REGION Network 18: Special characters — Common character widths and additional whitespace characters
   // ▀▀▀▀▀▀▀▀▀▀▀▀▀▀▀▀▀▀▀▀▀▀▀▀▀▀▀▀▀▀▀▀▀▀▀▀▀▀▀▀▀▀▀▀
   // 
   // TITLE:    COMMON CHARACTER WIDTHS AND ADDITIONAL WHITESPACE CHARACTERS
   // 
   // ▄▄▄▄▄▄▄▄▄▄▄▄▄▄▄▄▄▄▄▄▄▄▄▄▄▄▄▄▄▄▄▄▄▄▄▄▄▄▄▄▄▄▄▄
   // 
   // 
   // This section contains a list of the alphanumeric characters and common punctuation in terms of
   // character width (thinnest first).
   // 
   // The average character widths for each group are based on the frequency of letter usage in 
   // standard (British) English.
   // 
   // The additional whitespace characters complete the set of TIA Portal whitespace characters, these
   // are included for completeness, but duplicate the widths of the standard whitespace characters 
   // listed in previous sections.
   // 
   // 
   // 
   // ▄▄▄▄▄▄▄▄▄▄▄▄▄▄▄▄▄▄▄▄▄▄▄▄▄▄▄▄▄▄▄▄▄▄▄▄▄▄▄▄▄▄▄▄
   // NORMAL CHARACTERS BY WIDTH
   // 
   // 
   // ▐I▌1sp
   // ▐J▌1⅓ sp
   // ▐T▌1⅔ SP
   // ▐F▌2 sp
   // ▐L▌2 sp
   // ▐P▌2 sp
   // ▐R▌2 sp
   // ▐A▌2⅓ SP
   // ▐B▌2⅓ SP
   // ▐C▌2⅓ SP
   // ▐E▌2⅓3 SP
   // ▐K▌2⅓ SP
   // ▐S▌2⅓ SP
   // ▐V▌2⅓ SP
   // ▐X▌2⅓ SP
   // ▐Y▌2⅓ SP
   // ▐Z▌2⅓ SP
   // ▐D▌2⅔ sp
   // ▐G▌2⅔ sp
   // ▐H▌2⅔ sp
   // ▐N▌2⅔ sp
   // ▐U▌2⅔ sp
   // ▐M▌3 sp
   // ▐O▌3 sp
   // ▐Q▌3 sp
   // ▐W▌3 sp
   // Upper avg. (based on frequency and width) = 2.25 normal spaces
   // 
   // ▐f▌1 sp
   // ▐i▌1 sp
   // ▐j▌1 sp
   // ▐l▌1 sp
   // ▐r▌1⅓ sp
   // ▐t▌1⅓ sp
   // ▐x▌1⅔ sp
   // ▐y▌1⅔ sp
   // ▐z▌1⅔ sp
   // ▐c▌2 sp
   // ▐k▌2 sp
   // ▐s▌2 sp
   // ▐v▌2 sp
   // ▐a▌2⅓ sp
   // ▐b▌2⅓ sp
   // ▐d▌2⅓ sp
   // ▐e▌2⅓ sp
   // ▐g▌2⅓ sp
   // ▐h▌2⅓ sp
   // ▐n▌2⅓ sp
   // ▐o▌2⅓ sp
   // ▐p▌2⅓ sp
   // ▐q▌2⅓ sp
   // ▐u▌2⅓ sp
   // ▐w▌3 sp
   // ▐m▌3⅔ sp
   // Lower avg. (based on frequency and width) = 2.00 normal spaces
   // 
   // ▐0▌2⅓ sp
   // ▐1▌2⅓ sp
   // ▐2▌2⅓ sp
   // ▐3▌2⅓ sp
   // ▐4▌2⅓ sp
   // ▐5▌2⅓ sp
   // ▐6▌2⅓ sp
   // ▐7▌2⅓ sp
   // ▐8▌2⅓ sp
   // ▐9▌2⅓ sp
   // Numbers = 2.33 sp
   // 
   // ▐!▌1 sp
   // ▐'▌1 sp
   // ▐,▌1 sp
   // ▐-▌1 sp
   // ▐.▌1 sp
   // ▐/▌1 sp
   // ▐\▌1 sp
   // ▐|▌1 sp
   // ▐[▌1⅓ sp
   // ▐]▌1⅓ sp
   // ▐:▌1⅓ sp
   // ▐:▌1⅓ sp
   // ▐(▌1⅓ sp
   // ▐)▌1⅓ sp
   // ▐{▌1⅔ sp
   // ▐}▌1⅔ sp
   // ▐"▌1⅔ sp
   // ▐?▌1⅔ sp
   // ▐<▌2 sp
   // ▐>▌2 sp
   // ▐^▌2 sp
   // ▐_▌2 sp
   // ▐~▌2 sp
   // ▐=▌2⅓ sp
   // ▐$▌2⅓ sp
   // ▐*▌2⅓ sp
   // ▐+▌2⅓ sp
   // ▐`▌2⅓ sp
   // ▐&▌2⅔ sp
   // ▐#▌2⅔ sp
   // ▐%▌3 sp
   // ▐@▌3⅓ sp
   // Punctuation avg. 1 sp (based on comma, full stop and dash being the most common)
   // 
   // 
   // 
   // ▄▄▄▄▄▄▄▄▄▄▄▄▄▄▄▄▄▄▄▄▄▄▄▄▄▄▄▄▄▄▄▄▄▄▄▄▄▄▄▄▄▄▄▄
   // ALL OTHER WHITESPACE CHARACTERS
   // 
   // The other whitespace characters (Hair space, figure space &c.) are supported by the Siemens
   // font, but have the identical widths to those listed above. The full list is shown below:
   // 
   // ▐  ▌2 Em spaces
   // ▐    ▌4 En space      (1/2 em)
   // ▐      ▌6 Three per em     (1/3 em)
   // ▐        ▌8 Punctuation space (1/4 em)
   // ▐        ▌8 Normal space      (1/4 em)
   // ▐        ▌8 Four per em      (1/4 em)
   // ▐        ▌8 Figure space     (1/4 em)
   // ▐            ▌12 Six per em    (1/6 em)
   // ▐            ▌12 Hair space       (1/6 em)
   // 
   //                 ━━━  ⬙⬙⬙⬙⬙⬙  ━━━
   // 
   // 
   // ██████████████ █ █ █ █  END   █ █ █ █ ██████████████
END_REGION

REGION Network 19: OB1 NETWORK 1 — Project description
   // ▀▀▀▀▀▀▀▀▀▀▀▀▀▀▀▀▀▀▀▀▀▀▀▀▀▀▀▀▀▀▀▀▀▀▀▀▀▀▀▀▀▀▀▀
   // 
   // TITLE:    PS2001 — PRACTICAL SERIES AUTOMATION LIBRARY
   // 
   // ▄▄▄▄▄▄▄▄▄▄▄▄▄▄▄▄▄▄▄▄▄▄▄▄▄▄▄▄▄▄▄▄▄▄▄▄▄▄▄▄▄▄▄▄
   // 
   // 
   // ――――――――――――――――――――――――――――――――――
   // COPYRIGHT:       © 2020 Michael Gledhill
   //           Part of the Practical Series of Publications
   //           Published in the United Kingdom
   //           mg@practicalseries.com
   //           https://practicalseries.com
   // ――――――――――――――――――――――――――――――――――
   // CUSTOMER:       Practical Series of Publications (PSP)
   // 
   // PROJECT:      Practical Series Automation Library (PAL)
   // 
   // PROJECT NO.:       PS2001
   // ――――――――――――――――――――――――――――――――――
   // CONTROLLER:       CPU 1515-2PN/DP
   // 
   // CONTROLLER NAME:    CON100
   // 
   // IP ADDRESS:      192.168.001.100
   // ――――――――――――――――――――――――――――――――――
   // TIA PROJECT NAME:    PS2001-PAL-D0000
   // 
   // STATUS:        DEVELOPMENT
   // ――――――――――――――――――――――――――――――――――
   // PROTECTION:     To minimise the risk of inadvertent modification to 
   //           tested modules, certain blocks will be released for 
   //           use with “protected access” (referred to a “write 
   //           protection” in Siemens terminology), this allows the 
   //           block to be used normally, but prevents the block 
   //           being accidentally modified. 
   // 
   //           This is in accordance with the risk assessment given 
   //           in the Validation Plant (VP), Appendix A [Ref. 002].
   // 
   //           ┌─────────────────────┐
   //           │ THE WRITE PROTECTION PASSWORD IS: PS2001 │
   //           └─────────────────────┘
   // 
   // 
   // ▄▄▄▄▄▄▄▄▄▄▄▄▄▄▄▄▄▄▄▄▄▄▄▄▄▄▄▄▄▄▄▄▄▄▄▄▄▄▄▄▄▄▄▄
   // PROJECT OVERVIEW
   // 
   // 
   // The PAL is a library of software modules and templates that have been developed for the 
   // Siemens Simatic S7-1500 range of controllers (and to a lesser extent the S7-1200 range).
   // 
   // The full library and all necessary documentation is available from the Practical Series website:
   // 
   //      https://practicalseries.com/2001-pal/index.html
   // 
   // 
   // The PAL is configured and deployed using the Siemens Simatic TIA Portal programming 
   // environment.
   // 
   // The PAL software structure is designed such that it is applicable to virtually all industrial 
   // applications that can generally controlled by a programmable logic controller.
   // 
   // The PAL software being developed as part of this Project, is considered to be suitable for use in 
   // the following types of industries (this is not an exhaustive list):
   // 
   //    •   Water and waste water treatment
   //    •   Pharmaceutical and batch production
   //    •   Brewing and fermentation
   //    •   Chemical manufacturing
   //    •   Oil and gas systems
   //    •   Food and beverage production
   // 
   // Such applications can generally be thought of as processes that operate with a response time
   // of more than 100 ms. I.e. the system would not be expected to respond to some stimuli faster
   // than 100 ms. In practice, a Controller may (and usually will) respond faster than this; however, 
   // a response time of 100 ms is considered to be an acceptable limit for PLC control.
   // 
   // At its most basic level, the PAL will be a library of software modules that control the fundamental 
   // aspects of an industrial plant; such modules would for example read the value of an instrument, 
   // operate a valve or drive, perform a calculation &c.
   // 
   // Such software modules are referred to as standard modules, these are fixed modules that 
   // perform a particular function and are identical across all software installations.
   // 
   // The PAL also contains application specific modules; these contain software that is applicable 
   // to the plant being controlled.
   // 
   // The Practical Series Automation Library is freely available under the MIT Open Source licence 
   // (see below). Those who find it useful may, if they wish, make a donation to support the library. 
   // 
   // Donations can be made here:
   // 
   //      https://practicalseries.com/2001-pal/11-web/81-00-pay.html
   // 
   // The PAL contains fully deployable software that has been developed by the author in his 
   // profession as a chartered electrical engineer. It is currently in use on various live plants 
   // throughout the UK and in some other parts of the world. 
   // 
   // This software is suitable for controlling and automating most industrial applications (typical 
   // process applications). It is easy to use and configure, but does have a degree of practical 
   // complexity appropriate for the environments within which it is employed. It is heavily 
   // configurable, has various operating modes and is suitable for a multitude of industrial 
   // applications.
   // 
   // IF YOU DON’T UNDERSTAND IT, DON’T USE IT. IF YOU DO USE IT, YOU DO SO AT YOUR OWN RISK.
   // 
   //                ━━━   ⬙⬙⬙⬙⬙⬙   ━━━
   // 
   // ▄▄▄▄▄▄▄▄▄▄▄▄▄▄▄▄▄▄▄▄▄▄▄▄▄▄▄▄▄▄▄▄▄▄▄▄▄▄▄▄▄▄▄▄
   // DOCUMENT REFERENCES
   // 
   //  ――――――――――――――――――――――――――――――――――――――――――
   //  REF.     DOCUMENT NO.       TITLE
   //  ――――――――――――――――――――――――――――――――――――――――――
   //  001  PS2001-5-0101-001   Quality Plan (QP)
   //  002  PS2001-5-0121-002   Validation Plan (VP)
   //  003  PS2001-5-0131-003   Test Plan (TP)
   //  004  PS2001-5-1101-001   User requirements specification (URS)
   //  005  PS2001-5-1111-001   Requirement Traceability Matrix (RTM)
   //  006  PS2001-5-2101-001   Functional Specification (FS) 
   //  007  PS2001-5-2211-001   Hardware Design Specification (HDS)
   //  008  PS2001-5-2311-001   Software Design Specification (SDS)
   //  009  PS2001-5-7111-001   User Guide (UG)
   //  010  PS2001-5-2313-011   Style Guide (SG)
   //  011  PS2001-5-2312-fcNo.    Software Module Design Specification (SMDS)
   //  012  PS2001-5-2301-001   Software Module Register (SMR)
   //  013  PS2001-5-2302-011   Software Control and Mechanism (SCM)
   //  ――――――――――――――――――――――――――――――――――――――――――
   // 
   //                ━━━   ⬙⬙⬙⬙⬙⬙   ━━━
   // 
   // 
   // ▄▄▄▄▄▄▄▄▄▄▄▄▄▄▄▄▄▄▄▄▄▄▄▄▄▄▄▄▄▄▄▄▄▄▄▄▄▄▄▄▄▄▄▄
   // COMPLETED MODULES 
   // 
   // COMPLETED MODULES 
   // 
   //  ――――――――――――――――――――-―-- STATIC DATA       ― DYNAMIC  DAT A   ―
   //  BLOCK     NAME         REVISION    UDT/DB    REVISION  UDT/DB    REVISION  
   //  ――――――――――――――――――――――――――――――――――――――――――
   //  FC01001 StdSysGlobalData      001.000   UT 01000   001.000-R UT 21000   001.000-R
   //                  2020-11-20   UT 01001   001.000-R UT 21000   001.000-R 
   //                           None           DB21000   001.000-R
   //  ――――――――――――――――――――――――――――――――――――――――――
   //  FC02001 StdInstAnalogRead    001.000   UT 02001   001.000-R UT 22001   001.000-R
   //                  2020-11-20   DB02001   001.000-R DB22001   001.000-R
   //  ――――――――――――――――――――――――――――――――――――――――――
   //  FC18001 StdSubScaleAI      001.000   None           None 
   //                  2020-12-09   None           None
   //  ――――――――――――――――――――――――――――――――――――――――――
   //  FC18151 StdSubTimeEventRTC   001.000   None           UT 38151   001.000-R
   //                  2020-11-20                  DB38151   001.000-R
   //  ――――――――――――――――――――――――――――――――――――――――――
   //  FC61000 DocGenExample     001.000   None           None 
   //                  2020-11-20   None           None          
   //  ――――――――――――――――――――――――――――――――――――――――――
   //  FC21000 AppSys          001.000   None           None 
   //                  2020-12-04   None           None          
   //  ――――――――――――――――――――――――――――――――――――――――――
   //  See Software Module Register [Ref. 012] for full details
   // 
   //                ━━━   ⬙⬙⬙⬙⬙⬙   ━━━
   // 
   // 
   // ▀▀▀▀▀▀▀▀▀▀▀▀▀▀▀▀▀▀▀▀▀▀▀▀▀▀▀▀▀▀▀▀▀▀▀▀▀▀▀▀▀▀▀▀
   // LICENCE AND CONTACT INFORMATION
   // 
   // This software and its associated documentation is made available under the MIT Licence:
   // 
   // ════════════════════════════════════════════
   // 
   // The MIT License (MIT)
   // 
   // Copyright © 2020 Michael Gledhill
   // 
   // Permission is hereby granted, free of charge, to any person obtaining a copy of this software 
   // and associated documentation files (the “Software”), to deal in the Software without restriction, 
   // including without limitation the rights to use, copy, modify, merge, publish, distribute, 
   // sublicense, and/or sell copies of the Software, and to permit persons to whom the Software is 
   // furnished to do so, subject to the following conditions: 
   // 
   // The above copyright notice and this permission notice shall be included in all copies or 
   // substantial portions of the Software.
   // 
   // THE SOFTWARE IS PROVIDED “AS IS”, WITHOUT WARRANTY OF ANY KIND, EXPRESS OR IMPLIED, 
   // INCLUDING BUT NOT LIMITED TO THE WARRANTIES OF MERCHANTABILITY, FITNESS FOR A 
   // PARTICULAR PURPOSE AND NON-INFRINGEMENT. IN NO EVENT SHALL THE AUTHORS OR COPYRIGHT 
   // HOLDERS BE LIABLE FOR ANY CLAIM, DAMAGES OR OTHER LIABILITY, WHETHER IN AN ACTION OF 
   // CONTRACT, TORT OR OTHERWISE, ARISING FROM, OUT OF OR IN CONNECTION WITH THE SOFTWARE 
   // OR THE USE OR OTHER DEALINGS IN THE SOFTWARE.
   // 
   // ════════════════════════════════════════════
   //                    ┌────────────┐
   // You can reach the author by email here:   │  mg@practicalseries.com  │
   //                    └────────────┘
   // Questions, corrections, constructive criticism and complaints (polite ones) are invited.
   // 
   // ▄▄▄▄▄▄▄▄▄▄▄▄▄▄▄▄▄▄▄▄▄▄▄▄▄▄▄▄▄▄▄▄▄▄▄▄▄▄▄▄▄▄▄▄
   // 
   // 
   //                ━━━   ⬙⬙⬙⬙⬙⬙   ━━━
   // 
   // 
   // 
   // ██████████████ █ █ █ █  END   █ █ █ █ ██████████████
END_REGION

REGION Network 20: OB1 NETWORK 2 — Current revision and modification history
   // ▄▄▄▄▄▄▄▄▄▄▄▄▄▄▄▄▄▄▄▄▄▄▄▄▄▄▄▄▄▄▄▄▄▄▄▄▄▄▄▄▄▄▄▄
   // MODIFICATION HISTORY (GITHUB VERSION CONTROL SYSTEM)
   // 
   // 
   // This is a complete summary of all primary software modifications (commit points) made to this 
   // TIA Portal project (the latest commit tag is at the top of the list). 
   // 
   // The latest commit tag, author and the date of the revision are hardcoded into the Controller in 
   // this network (allowing revision data to be obtained directly from the Controller).
   // 
   // The development of the software project is stored and managed within the GIT Source Code 
   // Management system (a version control system or VCS) in conjunction with the GitHub online 
   // hosting system. The software in its entirety is available in the GitHub remote repository:
   // 
   //      https://github.com/practicalseries/PS2001-pal-software
   // 
   // This repository is public and can be freely “forked” (copied) and used under the MIT Licence.
   // The MIT Licence is reproduced in full in the previous network.
   // 
   //  ———————————————————————————————————————————
   //  DATE     COMMIT TAG       AUTHOR        REASON FOR MODIFICATION
   //  ———————————————————————————————————————————
   //  2021.02.02    D0002      M. Gledhill      Baseline build
   // 
   //  2021.02.02    D0001      M. Gledhill      Hardware build
   // 
   //  2021.02.02    D0000      M. Gledhill      Initial commit — repository created
   //  ———————————————————————————————————————————
   // 
   // 
   // ▄▄▄▄▄▄▄▄▄▄▄▄▄▄▄▄▄▄▄▄▄▄▄▄▄▄▄▄▄▄▄▄▄▄▄▄▄▄▄▄▄▄▄▄
   RUNG wire#powerrail
      I_Contact( #_FALSE )
      wire#w1
      S_Move(in := 'PS2001', out => #revInfo.REV_BLOCK)
   END_RUNG
   RUNG wire#w1
      S_Move(in := '001.000-R', out => #revInfo.REV_NUMBER)
   END_RUNG
   RUNG wire#w1
      S_Move(in := '2020.10.20', out => #revInfo.REV_DATE)
   END_RUNG
   RUNG wire#w1
      S_Move(in := 'M. Gledhill', out => #revInfo.REV_AUTHOR)
   END_RUNG
   // the same network as SCL:
   IF NOT #_FALSE THEN
       #revInfo.REV_BLOCK := 'PS2001';
       #revInfo.REV_NUMBER := '001.000-R';
       #revInfo.REV_DATE := '2020.10.20';
       #revInfo.REV_AUTHOR := 'M. Gledhill';
   END_IF;
END_REGION

REGION Network 21: Load the system RTC and store in local variable [typical network comment]
   // ▀▀▀▀▀▀▀▀▀▀▀▀▀▀▀▀▀▀▀▀▀▀▀▀▀▀▀▀▀▀▀▀▀▀▀▀▀▀▀▀▀▀▀▀
   // The system block RD_SYS_T reads the time of day, the date and the day of week from the system 
   // real time clock as a DTL (or Date_And_Time_Long) data type (one just being the shorthand 
   // notation of the other). The result is stored in a local variable for decoding.
   // 
   // The DTL data type stores the date and time information in 8 consecutive bytes in BCD format 
   // as follows:
   // 
   // 
   //  ――――――――――――――――――――――――――――――――――――――――――
   //  DATA         DESCRIPTION
   // 
   //  0          Dear        (00h-89h = 2000 to 2089)   (90h-99h = 1990 to 1999)
   //  1          Month      (00h-12h = Jan to Dec)
   //  2          Day       (01h-31h)
   //  3          Hour        (00h-23h)
   //  4          Minute        (00h-59h)
   //  5          Month      (00h-12h = Jan to Dec)
   //  6-7         Millisecond      Uses byte 6 and most significant 4 bits of byte 7)
   //  7          Day of Week    least significant 4 bits (1h-7h = Sun to Sat)
   //  ――――――――――――――――――――――――――――――――――――――――――
   // 
   // 
   // The local variable is of type DTL (Date_And_Time_Long), this is compatible with the DT output
   // from RD_SYST, but allows the individual elements of the DT structure to be accesses
   // individually as symbols.
   // 
   // Note:    The DTL format can store more information (it can for example handle years in the 
   //      range 1970 to 2262; however, it will still only store the data in the table above
   //      when used with RS_SYS_T. 
   // ▄▄▄▄▄▄▄▄▄▄▄▄▄▄▄▄▄▄▄▄▄▄▄▄▄▄▄▄▄▄▄▄▄▄▄▄▄▄▄▄▄▄▄▄
END_REGION

REGION Network 22: ██ STEP 03340 — DECLARATION (RUNNING) [sequence network comment]
   // ▀▀▀▀▀▀▀▀▀▀▀▀▀▀▀▀▀▀▀▀▀▀▀▀▀▀▀▀▀▀▀▀▀▀▀▀▀▀▀▀▀▀▀▀
   // 
   //  ███   ███   ███  █  █   ███  
   // █   █ █   █ █   █ █  █  █   █ 
   // █  ██     █     █ █  █  █  ██ 
   // █ █ █  ███   ███  █████ █ █ █ 
   // ██  █     █     █    █  ██  █ 
   // █   █ █   █ █   █    █  █   █ 
   //  ███   ███   ███     █   ███  
   // 
   // ▄▄▄▄▄▄▄▄▄▄▄▄▄▄▄▄▄▄▄▄▄▄▄▄▄▄▄▄▄▄▄▄▄▄▄▄▄▄▄▄▄▄▄▄
   // STEP DESCRIPTION
   // 
   // 
   // Open the dry air purge valve (SV4201), activate the operator prompt ABORT PURGE.
   // 
   // If the main chamber humidity level falls below the target value proceed to the next step.
   // 
   // If the operator presses the ABORT PURGE button proceed to step 03400.
   // 
   // 
   // 
   // ▄▄▄▄▄▄▄▄▄▄▄▄▄▄▄▄▄▄▄▄▄▄▄▄▄▄▄▄▄▄▄▄▄▄▄▄▄▄▄▄▄▄▄▄
   // STEP PHASE AND DELAY CONDITIONS
   // 
   // 
   //  ――――――――――――――――――――――――――――――――――――――――――
   //  PHASE         ACTION
   //  ――――――――――――――――――――――――――――――――――――――――――
   //  INITIALISING      Activate the ABORT PURGE enable signal
   // 
   //  PROCESSING    Open SV4201
   // 
   //  TERMINATING    Clear the ABORT PURGE enable signal and any ABORT PURGE pressed
   //           signal
   // 
   //  STEP DELAY      No delay
   //  ――――――――――――――――――――――――――――――――――――――――――
   // 
   // 
   // 
   // ▄▄▄▄▄▄▄▄▄▄▄▄▄▄▄▄▄▄▄▄▄▄▄▄▄▄▄▄▄▄▄▄▄▄▄▄▄▄▄▄▄▄▄▄
   // STEP TRANSITION CONDITIONS
   // 
   // 
   //  ――――――――――――――――――――――――――――――――――――――――――
   //  TRANSITION      TO STEP    TRANSITION CONDITIONS
   //  ――――――――――――――――――――――――――――――――――――――――――
   //  1.        03350      HIC001 ≤ HUMIDITY_LIMIT
   // 
   //  2.        03400      Operator has pressed ABORT PURGE button
   //  ――――――――――――――――――――――――――――――――――――――――――
   // 
   // 
   // ▄▄▄▄▄▄▄▄▄▄▄▄▄▄▄▄▄▄▄▄▄▄▄▄▄▄▄▄▄▄▄▄▄▄▄▄▄▄▄▄▄▄▄▄
END_REGION

REGION Network 23: STEP 03340 — ACTION (INITIALISE) [sequence network comment]
   // ▀▀▀▀▀▀▀▀▀▀▀▀▀▀▀▀▀▀▀▀▀▀▀▀▀▀▀▀▀▀▀▀▀▀▀▀▀▀▀▀▀▀▀▀
   // INITIALISE PHASE
   // 
   // Activate the ABORT PURGE enable signal
   // (this is a temporary signal passed to the handling DB at the end of the block)
   // ▄▄▄▄▄▄▄▄▄▄▄▄▄▄▄▄▄▄▄▄▄▄▄▄▄▄▄▄▄▄▄▄▄▄▄▄▄▄▄▄▄▄▄▄
END_REGION

REGION Network 24: STEP 03340 — TRANSITION 01 [sequence network comment]
   // ▀▀▀▀▀▀▀▀▀▀▀▀▀▀▀▀▀▀▀▀▀▀▀▀▀▀▀▀▀▀▀▀▀▀▀▀▀▀▀▀▀▀▀▀
   // TRANSITION CONDITION 01
   // 
   // Wait for humidity to reach target level HIC001 ≤ HUMIDITY_LIMIT
   // ▄▄▄▄▄▄▄▄▄▄▄▄▄▄▄▄▄▄▄▄▄▄▄▄▄▄▄▄▄▄▄▄▄▄▄▄▄▄▄▄▄▄▄▄
END_REGION

REGION Network 25: LICENCE AND CONTACT INFORMATION [final network]
   // ▀▀▀▀▀▀▀▀▀▀▀▀▀▀▀▀▀▀▀▀▀▀▀▀▀▀▀▀▀▀▀▀▀▀▀▀▀▀▀▀▀▀▀▀
   // LICENCE AND CONTACT INFORMATION
   // 
   // This software and its associated documentation is made available under the MIT Licence:
   // 
   // ════════════════════════════════════════════
   // 
   // The MIT License (MIT)
   // 
   // Copyright © 2020 Michael Gledhill
   // 
   // Permission is hereby granted, free of charge, to any person obtaining a copy of this software 
   // and associated documentation files (the “Software”), to deal in the Software without restriction, 
   // including without limitation the rights to use, copy, modify, merge, publish, distribute, 
   // sublicense, and/or sell copies of the Software, and to permit persons to whom the Software is 
   // furnished to do so, subject to the following conditions: 
   // 
   // The above copyright notice and this permission notice shall be included in all copies or 
   // substantial portions of the Software.
   // 
   // THE SOFTWARE IS PROVIDED “AS IS”, WITHOUT WARRANTY OF ANY KIND, EXPRESS OR IMPLIED, 
   // INCLUDING BUT NOT LIMITED TO THE WARRANTIES OF MERCHANTABILITY, FITNESS FOR A 
   // PARTICULAR PURPOSE AND NON-INFRINGEMENT. IN NO EVENT SHALL THE AUTHORS OR COPYRIGHT 
   // HOLDERS BE LIABLE FOR ANY CLAIM, DAMAGES OR OTHER LIABILITY, WHETHER IN AN ACTION OF 
   // CONTRACT, TORT OR OTHERWISE, ARISING FROM, OUT OF OR IN CONNECTION WITH THE SOFTWARE 
   // OR THE USE OR OTHER DEALINGS IN THE SOFTWARE.
   // 
   // ════════════════════════════════════════════
   //                    ┌────────────┐
   // You can reach the author by email here:   │  mg@practicalseries.com  │
   //                    └────────────┘
   // Questions, corrections, constructive criticism and complaints (polite ones) are invited.
   // 
   // ▄▄▄▄▄▄▄▄▄▄▄▄▄▄▄▄▄▄▄▄▄▄▄▄▄▄▄▄▄▄▄▄▄▄▄▄▄▄▄▄▄▄▄▄
   RUNG wire#powerrail
      I_Contact( #_FALSE )
      wire#w1
      S_Move(in := 'MIT LICENSE', out => #licInfo.LICENCE_TYPE)
   END_RUNG
   RUNG wire#w1
      S_Move(in := '2020 Michael Gledhill', out => #licInfo.COPYRIGHT)
   END_RUNG
   // the same network as SCL:
   IF NOT #_FALSE THEN
       #licInfo.LICENCE_TYPE := 'MIT LICENSE';
       #licInfo.COPYRIGHT := '2020 Michael Gledhill';
   END_IF;
END_REGION
END_FUNCTION
